(* CODESYS project State Machine.library
   Title: State Machine Twincat
   Version: 1.0.0.4
   Placeholder: State Machine Twincat
   Company: Home

Project tree, tasks and I/O mapping:
  libraries: Tc2_Standard, * (Beckhoff Automation GmbH); Tc2_System, * (Beckhoff Automation GmbH); Tc3_Module, * (Beckhoff Automation GmbH)
  DUTs/
    Actuators/
      TwoPos/
        data type E_TwoPosActuator_Fault
        data type E_TwoPosActuator_State
        data type ST_TwoPosActuator_Cfg
        data type ST_TwoPosActuator_HMI
        data type ST_TwoPosActuator_IO
        data type ST_TwoPosActuator_Sts
    Permissives/
      data type ST_PermIntlk_cfg
      data type ST_PermIntlk_HMI
      data type ST_PermIntlk_sts
    State Machine/
      data type E_SM_State
      data type SM_HMI
      data type SM_HMI_cfg
      data type SM_HMI_ocmd
      data type SM_HMI_sts
      data type ST_SM_Commands
      data type ST_SM_Conditions
      data type ST_SM_Internal
      data type ST_SM_PermissionGroups
      data type ST_SM_Permissions
      data type ST_SM_Status
      data type ST_SM_StepInfo
    Steps/
      data type ActiveStep
  GVLs/
  POUs/
    function block FB_Permissives [ST]
    function block FB_SequenceStep [ST]
    function block FB_StateMachine [ST]
    function block FB_TwoPosActuator [ST]
  VISUs/
*)

// DUTs/Actuators/TwoPos/E_TwoPosActuator_Fault
TYPE E_TwoPosActuator_Fault :
(
    None := 0,
    AdvanceTimeout := 1,
    RetractTimeout := 2,
    BothFeedbackOn := 3,
    UndefinedState := 4,
    PermissivesNotOK := 5,
    ConflictingCommands := 6,
    NoFeedback := 7
);
END_TYPE

// DUTs/Actuators/TwoPos/E_TwoPosActuator_State
TYPE E_TwoPosActuator_State :
(
    Undefined := 0,
    Retracted := 1,
    Advancing := 2,
    Advanced := 3,
    Retracting := 4,
    Fault := 5
);
END_TYPE

// DUTs/Actuators/TwoPos/ST_TwoPosActuator_Cfg
TYPE ST_TwoPosActuator_Cfg :
STRUCT
    cfgAdvTimeoutS : INT := 5;          // Advance timeout in seconds
    cfgRetTimeoutS : INT := 5;          // Retract timeout in seconds
    cfgHoldAtAdvanced : BOOL := FALSE;  // Hold valve energized when advanced
    cfgHoldAtRetracted : BOOL := FALSE; // Hold valve energized when retracted
END_STRUCT
END_TYPE

// DUTs/Actuators/TwoPos/ST_TwoPosActuator_HMI
TYPE ST_TwoPosActuator_HMI :
STRUCT
    // Status information for HMI
    sts : ST_TwoPosActuator_Sts;
    
    // Configuration from HMI
    cfg : ST_TwoPosActuator_Cfg;
    
    // Human-readable strings for HMI display
    stateString : STRING(80);      // Current state as text
    faultString : STRING(80);      // Current fault as text
    lastFaultString : STRING(80);  // Last fault as text
    
    // Operator commands from HMI
    ocmdAdvance : BOOL;         // Operator command to advance
    ocmdRetract : BOOL;         // Operator command to retract
    ocmdAllOff : BOOL;          // Operator command to turn all outputs off
    ocmdReset : BOOL;           // Operator command to reset fault
    
    // Permissive information for HMI
    advancePerms : ST_PermIntlk_HMI;  // Advance permissives
    retractPerms : ST_PermIntlk_HMI;  // Retract permissives
END_STRUCT
END_TYPE

// DUTs/Actuators/TwoPos/ST_TwoPosActuator_IO
TYPE ST_TwoPosActuator_IO :
STRUCT
    // Input feedbacks from field
    inFbkAdvanced AT %I* : BOOL;       // Advanced position feedback
    inFbkRetracted AT %I* : BOOL;      // Retracted position feedback
    
    // Output commands to field
    outValveAdvance AT %Q* : BOOL;     // Advance valve command
    outValveRetract AT %Q* : BOOL;     // Retract valve command
END_STRUCT
END_TYPE

// DUTs/Actuators/TwoPos/ST_TwoPosActuator_Sts
TYPE ST_TwoPosActuator_Sts :
STRUCT
    state : E_TwoPosActuator_State;     // Current state of actuator
    stsAdvanced : BOOL;                 // TRUE when actuator is advanced
    stsRetracted : BOOL;                // TRUE when actuator is retracted
    stsMoving : BOOL;                   // TRUE when actuator is in motion
    stsFaulted : BOOL;                  // TRUE when actuator is faulted
    faultCode : E_TwoPosActuator_Fault; // Current fault code
    lastFaultCode : E_TwoPosActuator_Fault; // Last fault code for diagnostics
    osAdvanced : BOOL;                  // One-shot when reaching advanced position
    osRetracted : BOOL;                 // One-shot when reaching retracted position
END_STRUCT
END_TYPE

// DUTs/Permissives/ST_PermIntlk_cfg
TYPE ST_PermIntlk_cfg :
STRUCT
    Name : STRING(80);                      // Name for the entire permissive set
    Desc : ARRAY [0..15] OF STRING(80);       // Descriptions for each bit
    BypassPermissives : INT;                  // Bypass bits: if a bit is 1, that permissive is bypassed
END_STRUCT
END_TYPE

// DUTs/Permissives/ST_PermIntlk_HMI
TYPE ST_PermIntlk_HMI :
STRUCT
	sts : ST_PermIntlk_sts;
	cfg : ST_PermIntlk_cfg;
END_STRUCT
END_TYPE

// DUTs/Permissives/ST_PermIntlk_sts
TYPE ST_PermIntlk_sts :
STRUCT
    PermIntlk : INT;    // Computed bitwise permissive status (each bit 1 = OK)
    OK        : BOOL;   // Overall status (TRUE if all required bits are OK)
END_STRUCT
END_TYPE

// DUTs/State Machine/E_SM_State
(* State Machine Enumeration *)
TYPE E_SM_State :
(
    STATE_IDLE := 0,
    STATE_RUNNING := 1,
    STATE_STOPPING := 2,
    STATE_HOMING := 4,
    STATE_ABORTING := 8,
    STATE_HOMED := 16,
    STATE_STOPPED := 32,
    STATE_ABORTED := 64,
    STATE_COMPLETE := 128,
    STATE_PAUSING := 256,
    STATE_PAUSED := 512,
    STATE_PROCEEDING := 1024
);
END_TYPE

// DUTs/State Machine/SM_HMI
TYPE SM_HMI :
STRUCT
  cfg : SM_HMI_cfg;
  ocmd : SM_HMI_ocmd;
  sts : SM_HMI_sts;
  NextStatePerms : ST_PermIntlk_HMI;
  ActiveStepHMI : ST_PermIntlk_HMI;
END_STRUCT
END_TYPE

// DUTs/State Machine/SM_HMI_cfg
TYPE SM_HMI_cfg :
STRUCT
  Name : STRING(40);
  HomePerm : ST_PermIntlk_HMI;
  StartPerm : ST_PermIntlk_HMI;
  ProceedPerm : ST_PermIntlk_HMI;
  AutoIntlk : ST_PermIntlk_HMI;
END_STRUCT
END_TYPE

// DUTs/State Machine/SM_HMI_ocmd
TYPE SM_HMI_ocmd :
STRUCT
  Abort : BOOL;
  Home : BOOL;
  Start : BOOL;
  Stop : BOOL;
  Pause : BOOL;
  Proceed : BOOL;
  Retry : BOOL;
  ActiveStatePermBypass : BOOL;
END_STRUCT
END_TYPE

// DUTs/State Machine/SM_HMI_sts
TYPE SM_HMI_sts :
STRUCT
  Automatic : BOOL;
  Manual : BOOL;
  StepMode : BOOL;
  Homing : BOOL;
  Homed : BOOL;
  Running : BOOL;
  Complete : BOOL;
  Stopping : BOOL;
  Stopped : BOOL;
  Aborting : BOOL;
  Aborted : BOOL;
  Pausing : BOOL;
  Paused : BOOL;
  Proceeding : BOOL;
  Faulted : BOOL;
  ChildFaulted : BOOL;
  ReadyToHome : BOOL;
  ReadyToProceed : BOOL;
  ReadyToStart : BOOL;
  AutoStartRequest : BOOL;
  AutoCycleRequest : BOOL;
  Blocked : BOOL;
  Starved : BOOL;
  Mode : DINT;
  Step : DINT;
  NextStep : DINT;
  ReturnNextStep : DINT;
END_STRUCT
END_TYPE

// DUTs/State Machine/ST_SM_Commands
(* Commands Structure - Groups all command inputs *)
TYPE ST_SM_Commands :
STRUCT
    Abort : BOOL;
    CompleteState : BOOL;
    Home : BOOL;
    Pause : BOOL;
    Proceed : BOOL;
    Retry : BOOL;
    Start : BOOL;
    Stop : BOOL;
END_STRUCT
END_TYPE

// DUTs/State Machine/ST_SM_Conditions
(* Conditions Structure - Groups process condition inputs *)
TYPE ST_SM_Conditions :
STRUCT
    Blocked : DINT;
    Starved : DINT;
END_STRUCT
END_TYPE

// DUTs/State Machine/ST_SM_Internal
(* Internal State Structure *)
TYPE ST_SM_Internal :
STRUCT
    PauseStep : ActiveStep;
    PreviousState : DINT;
    TimerReset : BOOL;
    LsOdd : DINT;
    ONS : DINT;
    StepHistoryMax : DINT;
END_STRUCT
END_TYPE

// DUTs/State Machine/ST_SM_PermissionGroups
(* Permission Group Handlers *)
TYPE ST_SM_PermissionGroups :
STRUCT
    AutoIntlk : ST_PermIntlk_HMI;
    HomePerm : ST_PermIntlk_HMI;
    ProceedPerm : ST_PermIntlk_HMI;
    StartPerm : ST_PermIntlk_HMI;
END_STRUCT
END_TYPE

// DUTs/State Machine/ST_SM_Permissions
(* Permissions Status Structure *)
TYPE ST_SM_Permissions :
STRUCT
    AutoIntlkOK : BOOL;
    HomePermOK : BOOL;
    ProceedPermOK : BOOL;
    StartPermOK : BOOL;
END_STRUCT
END_TYPE

// DUTs/State Machine/ST_SM_Status
(* Status Structure - Groups all status outputs *)
TYPE ST_SM_Status :
STRUCT
    Aborted : BOOL;
    Aborting : BOOL;
    ActiveState : BOOL;
    AutoCycleRequest : BOOL;
    Automatic : BOOL;
    AutoStartRequest : BOOL;
    Blocked : BOOL;
    Complete : BOOL;
    Faulted : BOOL;
    Homed : BOOL;
    Homing : BOOL;
    Manual : BOOL;
    Mode : DINT;
    Paused : BOOL;
    Pausing : BOOL;
    Proceeding : BOOL;
    ReadyToHome : BOOL;
    ReadyToProceed : BOOL;
    ReadyToStart : BOOL;
    Running : BOOL;
    Starved : BOOL;
    Stopped : BOOL;
    Stopping : BOOL;
    SubmoduleFaulted : BOOL;
    WaitingState : BOOL;
END_STRUCT
END_TYPE

// DUTs/State Machine/ST_SM_StepInfo
(* Step Information Structure *)
TYPE ST_SM_StepInfo :
STRUCT
    CurrentStep : DINT;
    NextStep : DINT;
    ReturnNextStep : DINT;
    ReturnState : DINT;  // Changed from enum to DINT for compatibility
    LastState : DINT;    // Changed from enum to DINT for compatibility
    CurrentState : DINT; // Changed from enum to DINT for compatibility
    StateString : STRING(40);
    StepTimerSeconds : REAL;
END_STRUCT
END_TYPE

// DUTs/Steps/ActiveStep
TYPE ActiveStep  :
STRUCT
  Step : DINT;
  StatusStepFaulted : BOOL;
  PermsHMI : ST_PermIntlk_cfg;
END_STRUCT
END_TYPE

// POUs/FB_Permissives
{attribute 'hide_all_locals'}
FUNCTION_BLOCK FB_Permissives
VAR_INPUT
    inPermissives : INT;           // Real-world permissive bits from hardware/sensors
    cfg           : ST_PermIntlk_cfg; // Configuration: name, bit descriptions, and bypass settings
END_VAR
VAR_OUTPUT PERSISTENT
    stsOK       : BOOL;            // Overall computed status (TRUE if all required permissives are OK)
    PermStatus  : INT;             // Bitwise computed permissive status (each bit set to 1 means that bit is OK)
END_VAR
VAR
    i         : INT;
    localStatus : INT;             // Local working variable for status
END_VAR

// Clear local status at start of each cycle
localStatus := 0;

// Loop over bits 0 to 15
FOR i := 0 TO 15 DO
    // Check if bypass is active for this bit (bypass bits are in cfg)
    IF (cfg.BypassPermissives AND SHL(1, i)) <> 0 THEN
        // Bypassed: treat this bit as OK
        localStatus := localStatus OR SHL(1, i);
    ELSE
        // Otherwise, if the real permissive bit is set, mark it as OK
        IF (inPermissives AND SHL(1, i)) <> 0 THEN
            localStatus := localStatus OR SHL(1, i);
        END_IF;
    END_IF;
END_FOR

// Save computed status to output variable
PermStatus := localStatus;

// Overall status: if all 16 bits are OK then stsOK is TRUE.
stsOK := (localStatus = -1);

END_FUNCTION_BLOCK

// POUs/FB_SequenceStep
{attribute 'hide_all_locals'}
FUNCTION_BLOCK FB_SequenceStep
VAR_INPUT
    inpStep              : DINT;  // Current step number (from sequence controller)
    cfgStep              : DINT;  // This FB's step number (step ID)
    cfgNextStep          : DINT;  // Next step if permissives are OK
    inpStepTimerSeconds  : DINT;  // Step timer value (managed externally)
    inpRetry             : BOOL;  // External retry command (to reset fault)
    inpStepPermissives   : INT;   // Actual permissive bits (from sensors, PLC, etc.)
    cfgStepTimeout       : INT;   // Timeout configuration (in seconds)
	inpFaultStep         : BOOL;  // Fault conditions outside of timeout 
END_VAR

VAR_IN_OUT
    ActiveStep           : ActiveStep; 
    // ActiveStep holds:
    //   Step              : DINT;  (current step number)
    //   StatusStepFaulted : BOOL;  (fault flag)
    //   PermsHMI          : ST_PermIntlk_cfg; (permissive configuration: Name, Desc, BypassPermissives)
END_VAR

VAR_OUTPUT
    outStepActive         : BOOL;  // TRUE when this step is active
    outStepActiveOS       : BOOL;  // One-shot rising pulse when step becomes active
    outFaultedStepActive  : BOOL;  // TRUE when this step is faulted
    outFaultedStepActiveOS: BOOL;  // One-shot rising pulse when a fault occurs
    outActiveStepTimedOut : BOOL;  // TRUE when the step times out
    outNextStep           : DINT;  // The next step number in sequence
END_VAR

VAR
    Step_P_Perm    : FB_Permissives; // Instance for permissives check
    rTrig_Activate : R_TRIG;         // Rising edge detector for step activation
    rTrig_Fault    : R_TRIG;         // Rising edge detector for fault detection
    rTrig_Retry    : R_TRIG;         // Rising edge detector for retry detection
END_VAR

// 1. Evaluate Permissives using FB_Permissives
Step_P_Perm.inPermissives := inpStepPermissives;
Step_P_Perm.cfg           := ActiveStep.PermsHMI;
Step_P_Perm();  // Execute permissives check

// 2. Update the ActiveStep with the current step
ActiveStep.Step := inpStep;

// 3. Determine if this step is active (active when inpStep equals cfgStep)
outStepActive := (inpStep = cfgStep);

// 4. Generate a one-shot pulse for step activation (rising edge)
rTrig_Activate.CLK := outStepActive;
rTrig_Activate();
outStepActiveOS := rTrig_Activate.Q;


// 5. Timeout Handling: If the externally managed timer exceeds the configured timeout, flag as timed out
IF 
(cfgStepTimeout <> 0 ) AND // cfgStepTimeout = 0 for no timeout fault
(inpStepTimerSeconds > cfgStepTimeout) 
THEN
    outActiveStepTimedOut := TRUE;
ELSE
    outActiveStepTimedOut := FALSE;
END_IF;

// 6. Fault Condition:
// A fault occurs if the step is active, the step has timed out, and the permissives are NOT OK.
IF outStepActive AND outActiveStepTimedOut AND (NOT Step_P_Perm.stsOK) 
OR inpFaultStep
THEN
    ActiveStep.StatusStepFaulted := TRUE;
END_IF;

// 7. Set the fault output based on the ActiveStep fault status
outFaultedStepActive := ActiveStep.StatusStepFaulted;

// 8. Generate a one-shot pulse for fault detection (rising edge)
rTrig_Fault.CLK := outFaultedStepActive;
rTrig_Fault();
outFaultedStepActiveOS := rTrig_Fault.Q;

// 9. Retry Logic: if a retry command is detected (rising edge on inpRetry) while faulted, clear the fault flag
rTrig_Retry.CLK := inpRetry;
rTrig_Retry();
IF rTrig_Retry.Q AND outFaultedStepActive THEN
    ActiveStep.StatusStepFaulted := FALSE;
END_IF;

// 10. Determine the next step:
// - If the step is faulted, set outNextStep to cfgStep + 1 (fault-handling step).
// - Else if the permissives are OK and the step is active, set outNextStep to cfgNextStep.
// - Otherwise, remain on the current step.
IF outFaultedStepActive THEN
    outNextStep := cfgStep + 1;
ELSIF Step_P_Perm.stsOK AND outStepActive THEN
    outNextStep := cfgNextStep;
ELSE
    outNextStep := inpStep;
END_IF;

END_FUNCTION_BLOCK

// POUs/FB_StateMachine
{attribute 'hide_all_locals'} // Hides all local variables
FUNCTION_BLOCK FB_StateMachine
VAR_INPUT
    EnableIn : BOOL;                     // Enable input for the function block
    cfgAutoRun : BOOL;                   // Configuration for auto-run capability
    inpAutoIntlk : INT := -1;            // Auto interlock input bits
    inpBlockedCondition : DINT;          // Blocked condition input
    inpHomePerm : INT := -1;             // Home permission input bits
    inpProceedPerm : INT := -1;          // Proceed permission input bits
    inpStartPerm : INT := -1;            // Start permission input bits
    inpStarvedCondition : DINT;          // Starved condition input
    inpSubmoduleFaulted : BOOL;          // Submodule fault indicator
END_VAR

VAR_OUTPUT
    EnableOut : BOOL;                    // Enable output for the function block
    outRetry : BOOL;                     // Retry output signal
    Status : ST_SM_Status;               // Status outputs (grouped)
    Permissions : ST_SM_Permissions;     // Permission status outputs (grouped)
    StepInfo : ST_SM_StepInfo;           // Step information (grouped)
    ConditionStatus : ST_SM_Conditions;  // Condition status (grouped)
END_VAR

VAR CONSTANT
    internalClearStep : ActiveStep;      // Constant for clearing a step
    EmptyHMIPerm : ST_PermIntlk_HMI;     // Empty HMI permissions structure
    
    // State constants
    STATE_IDLE : INT := 0;
    STATE_RUNNING : INT := 1;
    STATE_STOPPING : INT := 2;
    STATE_HOMING : INT := 4;
    STATE_ABORTING : INT := 8;
    STATE_HOMED : INT := 16;
    STATE_STOPPED : INT := 32;
    STATE_ABORTED : INT := 64;
    STATE_COMPLETE : INT := 128;
    STATE_PAUSING : INT := 256;
    STATE_PAUSED : INT := 512;
    STATE_PROCEEDING : INT := 1024;

    // Step range constants for sequence inference
    HOMING_MIN   : DINT := 1000; HOMING_MAX   : DINT := 1999;
    RUNNING_MIN  : DINT := 3000; RUNNING_MAX  : DINT := 3999;
    STOPPING_MIN : DINT := 2000; STOPPING_MAX : DINT := 2999;
    ABORTING_MIN : DINT := 5000; ABORTING_MAX : DINT := 5999;
    PAUSING_MIN  : DINT := 4000; PAUSING_MAX  : DINT := 4999;
    PROCEEDING_MIN : DINT := 6000; PROCEEDING_MAX : DINT := 6999;
END_VAR

VAR
    // Command request tracking
    CommandsRequested : ST_SM_Commands;  // Track command requests
    RetryComplete : BOOL;                // Flag for retry completion
    
    // Timer
    StepTimer : TON;                     // Step timer
    
    // Edge detection for commands
    R_TRIG_1 : R_TRIG;                  // For step transition
    R_TRIG_2 : R_TRIG;                  // For command retry
    R_TRIG_3 : R_TRIG;                  // For HMI retry
    R_TRIG_4 : R_TRIG;                  // For state transitions
    R_TRIG_5 : R_TRIG;                  // For sequence complete inference
    
    // Internal state tracking
    PauseStep : ActiveStep;              // Store step during pause
    PreviousState : DINT;                // Previous state
    PreviousStep : DINT;                 // Previous step for reference
    TimerReset : BOOL;                   // Flag to reset timer
    LsOdd : DINT;                        // Odd step check for fault detection
    ONS : DINT;                          // General one-shot
    StepHistoryMax : DINT;               // Step history maximum
    ReturnState : DINT;                  // Return state after pause
    ReturnNextStep : DINT;               // Return next step after pause
    
    // Permission handlers
    internalAutoIntlk : FB_Permissives;       // Auto interlock handler
    internalHomePerm : FB_Permissives;        // Home permission handler
    internalProceedPerm : FB_Permissives;     // Proceed permission handler
    internalStartPerm : FB_Permissives;       // Start permission handler
    
    // Configuration for permission handlers
    homePermCfg : ST_PermIntlk_cfg;      // Configuration for home permission handler
    startPermCfg : ST_PermIntlk_cfg;     // Configuration for start permission handler
    proceedPermCfg : ST_PermIntlk_cfg;   // Configuration for proceed permission handler
    autoIntlkCfg : ST_PermIntlk_cfg;     // Configuration for auto interlock handler
    
    // HMI data structures for permissions
    internalAutoIntlk_HMI : ST_PermIntlk_HMI;  // Auto interlock HMI structure
    internalHomePerm_HMI : ST_PermIntlk_HMI;   // Home permission HMI structure
    internalProceedPerm_HMI : ST_PermIntlk_HMI; // Proceed permission HMI structure
    internalStartPerm_HMI : ST_PermIntlk_HMI;  // Start permission HMI structure
    
    // Temp variables for step detection
    stepIsZero : BOOL;                   // Flag for zero step
    retryCmdActive : BOOL;               // Flag for retry command
    retryHmiActive : BOOL;               // Flag for HMI retry
    transitionActive : BOOL;             // Flag for state transition
    seqDone : BOOL;                      // Inferred sequence completion
END_VAR

VAR_IN_OUT 
    HMI : SM_HMI;                        // HMI interface
    CurrentStep : ActiveStep;            // Current active step
	NextStep : DINT;                     // Next step to transition to
	Commands : ST_SM_Commands;           // Command inputs (grouped)
END_VAR


//-----------------------------------------------------------------------------
// Main Implementation
//-----------------------------------------------------------------------------
EnableOut := EnableIn;

// Only execute if enabled
IF EnableIn THEN
    //-------------------------------------------------------------------------
    // Process permissions for different states
    //-------------------------------------------------------------------------
    
    // Update configuration from HMI
    homePermCfg := internalHomePerm_HMI.cfg;
    startPermCfg := internalStartPerm_HMI.cfg;
    proceedPermCfg := internalProceedPerm_HMI.cfg;
    autoIntlkCfg := internalAutoIntlk_HMI.cfg;
    
    // Home permission evaluation
    internalHomePerm(
        inPermissives := inpHomePerm,
        cfg := homePermCfg
    );
    Permissions.HomePermOK := internalHomePerm.stsOK;
    internalHomePerm_HMI.sts.OK := internalHomePerm.stsOK;
    internalHomePerm_HMI.sts.PermIntlk := internalHomePerm.PermStatus;
    
    // Start permission evaluation
    internalStartPerm(
        inPermissives := inpStartPerm,
        cfg := startPermCfg
    );
    Permissions.StartPermOK := internalStartPerm.stsOK;
    internalStartPerm_HMI.sts.OK := internalStartPerm.stsOK;
    internalStartPerm_HMI.sts.PermIntlk := internalStartPerm.PermStatus;
    
    // Proceed permission evaluation
    internalProceedPerm(
        inPermissives := inpProceedPerm,
        cfg := proceedPermCfg
    );
    Permissions.ProceedPermOK := internalProceedPerm.stsOK;
    internalProceedPerm_HMI.sts.OK := internalProceedPerm.stsOK;
    internalProceedPerm_HMI.sts.PermIntlk := internalProceedPerm.PermStatus;
    
    // Auto interlock evaluation
    internalAutoIntlk(
        inPermissives := inpAutoIntlk,
        cfg := autoIntlkCfg
    );
    Permissions.AutoIntlkOK := internalAutoIntlk.stsOK;
    internalAutoIntlk_HMI.sts.OK := internalAutoIntlk.stsOK;
    internalAutoIntlk_HMI.sts.PermIntlk := internalAutoIntlk.PermStatus;
    
    //-------------------------------------------------------------------------
    // Ready state calculations
    //-------------------------------------------------------------------------
    
    // Ready to Home: Stopped or Aborted + Home permissions OK + Auto interlock OK
    Status.ReadyToHome := (Status.Stopped OR Status.Aborted) AND 
                          Permissions.HomePermOK AND 
                          Permissions.AutoIntlkOK;
    
    // Ready to Start: (Homed or Complete) + Start permissions OK + Auto interlock OK + Not auto-start requested
    Status.ReadyToStart := (Status.Homed OR Status.Complete) AND 
                          Permissions.StartPermOK AND 
                          Permissions.AutoIntlkOK AND 
                          NOT Status.AutoStartRequest;
    
    // Ready to Proceed: Paused + Proceed permissions OK + Auto interlock OK
    Status.ReadyToProceed := Status.Paused AND 
                            Permissions.ProceedPermOK AND 
                            Permissions.AutoIntlkOK;

    //-------------------------------------------------------------------------
    // Clear Active Step if in waiting state
    //-------------------------------------------------------------------------
    IF Status.Homed OR Status.Complete OR Status.Stopped OR Status.Aborted THEN
        CurrentStep := internalClearStep;
    END_IF;
    
    // Clear pause step on proceeding or aborting
    transitionActive := Status.Proceeding OR Status.Aborting;
    R_TRIG_4(CLK := transitionActive);
    IF R_TRIG_4.Q THEN
        PauseStep := internalClearStep;
    END_IF;
    
    //-------------------------------------------------------------------------
    // Auto-start request logic
    //-------------------------------------------------------------------------
    
    // Auto start request handling
    Status.AutoStartRequest := CommandsRequested.Start AND NOT Permissions.StartPermOK;
    
    // Auto cycle request for auto-run when complete
    Status.AutoCycleRequest := cfgAutoRun AND Status.Complete AND NOT Permissions.StartPermOK;
    
    //-------------------------------------------------------------------------
    // Remember last state before change
    //-------------------------------------------------------------------------
    PreviousState := StepInfo.CurrentState;
    
    //-------------------------------------------------------------------------
    // Process command requests
    //-------------------------------------------------------------------------
    
    // Complete State Request
    IF Commands.CompleteState THEN
        CommandsRequested.CompleteState := TRUE;
        Commands.CompleteState := FALSE;  // Reset command
        // Clear other requests
        CommandsRequested.Start := FALSE;
        CommandsRequested.Abort := FALSE;
        CommandsRequested.Pause := FALSE;
        CommandsRequested.Home := FALSE;
        CommandsRequested.Proceed := FALSE;
        CommandsRequested.Stop := FALSE;
    END_IF;
    
    // Start Request
    IF Commands.Start OR HMI.ocmd.Start THEN
        IF Permissions.AutoIntlkOK AND Permissions.StartPermOK AND (Status.Homed OR Status.Complete) THEN
            CommandsRequested.Start := TRUE;
        END_IF;
        
        IF CommandsRequested.Start AND (Status.Homed OR Status.Complete OR Status.Stopped) OR Status.AutoStartRequest THEN
            CommandsRequested.Start := TRUE;
        END_IF;
        
        // Clear command signals
        IF Commands.Start THEN
            Commands.Start := FALSE;
        END_IF;
        
        IF HMI.ocmd.Start THEN
            HMI.ocmd.Start := FALSE;
        END_IF;
    END_IF;
    
    // Clear other requests if Start is requested
    IF CommandsRequested.Start THEN
        CommandsRequested.Abort := FALSE;
        CommandsRequested.Pause := FALSE;
        CommandsRequested.Home := FALSE;
        CommandsRequested.Proceed := FALSE;
        CommandsRequested.Stop := FALSE;
        CommandsRequested.CompleteState := FALSE;
    END_IF;
    
    // Auto-run handling
    IF cfgAutoRun AND Permissions.AutoIntlkOK AND Permissions.StartPermOK AND Status.Complete THEN
        CommandsRequested.Start := TRUE;
    END_IF;
    
    // Home Request
    IF Commands.Home OR HMI.ocmd.Home THEN
        IF (Status.Stopped OR Status.Aborted) AND Permissions.HomePermOK AND Permissions.AutoIntlkOK THEN
            CommandsRequested.Home := TRUE;
        END_IF;
        
        // Clear other requests
        CommandsRequested.Abort := FALSE;
        CommandsRequested.Pause := FALSE;
        CommandsRequested.Proceed := FALSE;
        CommandsRequested.Start := FALSE;
        CommandsRequested.Stop := FALSE;
        CommandsRequested.CompleteState := FALSE;
        
        // Clear command signals
        IF Commands.Home THEN
            Commands.Home := FALSE;
        END_IF;
        
        IF HMI.ocmd.Home THEN
            HMI.ocmd.Home := FALSE;
        END_IF;
    END_IF;
    
    // Pause Request
    IF Commands.Pause OR HMI.ocmd.Pause THEN
        CommandsRequested.Pause := TRUE;
        
        // Clear other requests
        CommandsRequested.Abort := FALSE;
        CommandsRequested.Home := FALSE;
        CommandsRequested.Proceed := FALSE;
        CommandsRequested.Start := FALSE;
        CommandsRequested.Stop := FALSE;
        CommandsRequested.CompleteState := FALSE;
        
        // Clear command signals
        IF Commands.Pause THEN
            Commands.Pause := FALSE;
        END_IF;
        
        IF HMI.ocmd.Pause THEN
            HMI.ocmd.Pause := FALSE;
        END_IF;
    END_IF;
    
    // Proceed Request
    IF Commands.Proceed OR HMI.ocmd.Proceed THEN
        IF Permissions.ProceedPermOK AND Permissions.AutoIntlkOK THEN
            CommandsRequested.Proceed := TRUE;
        END_IF;
        
        // Clear other requests
        CommandsRequested.Abort := FALSE;
        CommandsRequested.Home := FALSE;
        CommandsRequested.Pause := FALSE;
        CommandsRequested.Start := FALSE;
        CommandsRequested.Stop := FALSE;
        CommandsRequested.CompleteState := FALSE;
        
        // Clear command signals
        IF Commands.Proceed THEN
            Commands.Proceed := FALSE;
        END_IF;
        
        IF HMI.ocmd.Proceed THEN
            HMI.ocmd.Proceed := FALSE;
        END_IF;
    END_IF;
    
    // Stop Request
    IF Commands.Stop OR HMI.ocmd.Stop THEN
        CommandsRequested.Stop := TRUE;
        
        // Clear other requests
        CommandsRequested.Abort := FALSE;
        CommandsRequested.Home := FALSE;
        CommandsRequested.Proceed := FALSE;
        CommandsRequested.Start := FALSE;
        CommandsRequested.Pause := FALSE;
        CommandsRequested.CompleteState := FALSE;
        
        // Clear command signals
        IF Commands.Stop THEN
            Commands.Stop := FALSE;
        END_IF;
        
        IF HMI.ocmd.Stop THEN
            HMI.ocmd.Stop := FALSE;
        END_IF;
    END_IF;
    
    // Abort Request
    IF Commands.Abort OR HMI.ocmd.Abort THEN
        CommandsRequested.Abort := TRUE;
        
        // Clear other requests
        CommandsRequested.Stop := FALSE;
        CommandsRequested.Home := FALSE;
        CommandsRequested.Proceed := FALSE;
        CommandsRequested.Start := FALSE;
        CommandsRequested.Pause := FALSE;
        CommandsRequested.CompleteState := FALSE;
        
        // Clear command signals
        IF Commands.Abort THEN
            Commands.Abort := FALSE;
        END_IF;
        
        IF HMI.ocmd.Abort THEN
            HMI.ocmd.Abort := FALSE;
        END_IF;
    END_IF;
    
    //-------------------------------------------------------------------------
    // Sequence completion inference
    //-------------------------------------------------------------------------
    // If in an active state with a defined sequence range and the sequence
    // drives NextStep to 0 while the current step is within that state's
    // range, infer completion and trigger CompleteState internally.
    seqDone := FALSE;
    IF Status.Homing THEN
        seqDone := (StepInfo.CurrentStep >= HOMING_MIN) AND (StepInfo.CurrentStep <= HOMING_MAX) AND (NextStep = 0);
    ELSIF Status.Running THEN
        seqDone := (StepInfo.CurrentStep >= RUNNING_MIN) AND (StepInfo.CurrentStep <= RUNNING_MAX) AND (NextStep = 0);
    ELSIF Status.Stopping THEN
        seqDone := (StepInfo.CurrentStep >= STOPPING_MIN) AND (StepInfo.CurrentStep <= STOPPING_MAX) AND (NextStep = 0);
    ELSIF Status.Aborting THEN
        seqDone := (StepInfo.CurrentStep >= ABORTING_MIN) AND (StepInfo.CurrentStep <= ABORTING_MAX) AND (NextStep = 0);
    ELSIF Status.Pausing THEN
        seqDone := (StepInfo.CurrentStep >= PAUSING_MIN) AND (StepInfo.CurrentStep <= PAUSING_MAX) AND (NextStep = 0);
    ELSIF Status.Proceeding THEN
        seqDone := (StepInfo.CurrentStep >= PROCEEDING_MIN) AND (StepInfo.CurrentStep <= PROCEEDING_MAX) AND (NextStep = 0);
    END_IF;

    R_TRIG_5(CLK := seqDone);
    IF R_TRIG_5.Q THEN
        CommandsRequested.CompleteState := TRUE;
    END_IF;

    //-------------------------------------------------------------------------
    // State Transitions
    //-------------------------------------------------------------------------

    // Complete to Homed
    IF CommandsRequested.CompleteState AND Status.Homing THEN
        NextStep := 0;
        StepInfo.CurrentState := STATE_HOMED;
        CommandsRequested.CompleteState := FALSE;  // Clear after transition
    END_IF;
    
    // Running to Complete
    IF CommandsRequested.CompleteState AND Status.Running THEN
        NextStep := 0;
        StepInfo.CurrentState := STATE_COMPLETE;
        CommandsRequested.CompleteState := FALSE;  // Clear after transition
    END_IF;
    
    // Running to Stopping
    IF CommandsRequested.Stop AND Status.Running THEN
        StepInfo.CurrentState := STATE_STOPPING;
    END_IF;
    
    // Stopping to Stopped
    IF CommandsRequested.CompleteState AND Status.Stopping THEN
        NextStep := 0;
        StepInfo.CurrentState := STATE_STOPPED;
        CommandsRequested.CompleteState := FALSE;  // Clear after transition
    END_IF;
    
    // Aborting to Aborted
    IF CommandsRequested.CompleteState AND Status.Aborting THEN
        NextStep := 0;
        StepInfo.CurrentState := STATE_ABORTED;
        CommandsRequested.CompleteState := FALSE;  // Clear after transition
    END_IF;
    
    // Active State to Pausing
    // Handle state transitions to Pausing and remember the state to return to
    IF CommandsRequested.Pause AND (
        Status.Homing OR Status.Stopping OR Status.Aborting OR 
        Status.Homed OR Status.Complete OR Status.Proceeding OR Status.Running) THEN
        
        // Remember the current state and next step for later return
        IF NOT (Status.Homed OR Status.Complete OR Status.Proceeding) THEN
            ReturnState := StepInfo.CurrentState;
            ReturnNextStep := NextStep;
        END_IF;
        
        // Save the current step for paused state
        IF NOT (Status.Homed OR Status.Complete OR Status.Proceeding) THEN
            PauseStep := CurrentStep;
        ELSE
            PauseStep := internalClearStep;
        END_IF;
        
        // Transition to pausing state
        StepInfo.CurrentState := STATE_PAUSING;
        NextStep := 0;
    END_IF;
    
    // Pausing to Paused
    IF CommandsRequested.CompleteState AND Status.Pausing THEN
        NextStep := 0;
        StepInfo.CurrentState := STATE_PAUSED;
        CommandsRequested.CompleteState := FALSE;  // Clear after transition
    END_IF;
    
    // Proceeding to Step before Pausing
    IF CommandsRequested.CompleteState AND Status.Proceeding THEN
        CurrentStep := PauseStep;
        NextStep := ReturnNextStep;
        StepInfo.CurrentState := ReturnState;
        CommandsRequested.CompleteState := FALSE;  // Clear after transition
    END_IF;
    
    // Homed to Running
    IF (CommandsRequested.Start OR 
        (Status.AutoStartRequest AND Permissions.StartPermOK AND Permissions.AutoIntlkOK)) AND 
        (Status.Homed OR Status.Complete) THEN
        
        NextStep := 0;
        StepInfo.CurrentState := STATE_RUNNING;
        CommandsRequested.Start := FALSE;
    END_IF;
    
    // Homed to Stopped
    IF CommandsRequested.Stop AND Status.Homed THEN
        NextStep := 0;
        StepInfo.CurrentState := STATE_STOPPED;
    END_IF;
    
    // Complete to Stopped
    IF CommandsRequested.Stop AND Status.Complete THEN
        NextStep := 0;
        StepInfo.CurrentState := STATE_STOPPED;
    END_IF;
    
    // Stopped or Aborted to Homing
    IF CommandsRequested.Home AND (Status.Stopped OR Status.Aborted) THEN
        NextStep := 0;
        StepInfo.CurrentState := STATE_HOMING;
    END_IF;
    
    // Paused to Proceeding
    IF CommandsRequested.Proceed AND Status.Paused THEN
        NextStep := 0;
        StepInfo.CurrentState := STATE_PROCEEDING;
    END_IF;
    
    // Abort (from any state except Stopped/Aborted/Aborting)
    IF CommandsRequested.Abort AND NOT (Status.Stopped OR Status.Aborted OR Status.Aborting) THEN
        NextStep := 0;
        StepInfo.CurrentState := STATE_ABORTING;
    END_IF;
    
    //-------------------------------------------------------------------------
    // Save last state when changing
    //-------------------------------------------------------------------------
    IF StepInfo.CurrentState <> PreviousState THEN
        StepInfo.LastState := PreviousState;
    END_IF;
    
    //-------------------------------------------------------------------------
    // Update status flags based on current state
    //-------------------------------------------------------------------------
    // Reset all status flags first
    Status.Running := FALSE;
    Status.Stopping := FALSE;
    Status.Homing := FALSE;
    Status.Aborting := FALSE;
    Status.Homed := FALSE;
    Status.Stopped := FALSE;
    Status.Aborted := FALSE;
    Status.Complete := FALSE;
    Status.Pausing := FALSE;
    Status.Paused := FALSE;
    Status.Proceeding := FALSE;
    
    // Set corresponding status flag based on current state
    CASE StepInfo.CurrentState OF
        STATE_RUNNING:
            Status.Running := TRUE;
            StepInfo.StateString := 'Running';
        
        STATE_STOPPING:
            Status.Stopping := TRUE;
            StepInfo.StateString := 'Stopping';
        
        STATE_HOMING:
            Status.Homing := TRUE;
            StepInfo.StateString := 'Homing';
        
        STATE_ABORTING:
            Status.Aborting := TRUE;
            StepInfo.StateString := 'Aborting';
        
        STATE_HOMED:
            Status.Homed := TRUE;
            StepInfo.StateString := 'Homed';
        
        STATE_STOPPED:
            Status.Stopped := TRUE;
            StepInfo.StateString := 'Stopped';
        
        STATE_ABORTED:
            Status.Aborted := TRUE;
            StepInfo.StateString := 'Aborted';
        
        STATE_COMPLETE:
            Status.Complete := TRUE;
            StepInfo.StateString := 'Complete';
        
        STATE_PAUSING:
            Status.Pausing := TRUE;
            StepInfo.StateString := 'Pausing';
        
        STATE_PAUSED:
            Status.Paused := TRUE;
            StepInfo.StateString := 'Paused';
        
        STATE_PROCEEDING:
            Status.Proceeding := TRUE;
            StepInfo.StateString := 'Proceeding';
    END_CASE;
    
    // Set the active/waiting state flags
    Status.WaitingState := Status.Homed OR Status.Complete OR Status.Stopped OR Status.Paused OR Status.Aborted;
    Status.ActiveState := Status.Homing OR Status.Running OR Status.Stopping OR Status.Pausing OR Status.Proceeding OR Status.Aborting;
    
    // Set mode (0 = Manual, 1 = Automatic)
    IF Status.Stopped OR Status.Aborted OR Status.Paused THEN
        Status.Mode := 0;
        Status.Manual := TRUE;
        Status.Automatic := FALSE;
    ELSE
        Status.Mode := 1;
        Status.Manual := FALSE;
        Status.Automatic := TRUE;
    END_IF;

    //-------------------------------------------------------------------------
    // Step and timer management
    //-------------------------------------------------------------------------
    
    // Clear ActiveStep when transitioning to step 0 (when step becomes zero)
    stepIsZero := (StepInfo.CurrentStep = 0);
    R_TRIG_1(CLK := stepIsZero);
    IF R_TRIG_1.Q THEN
        CurrentStep := internalClearStep;
        // Also reset timer when entering step 0 (state transitions)
        TimerReset := TRUE;
        StepTimer(IN := FALSE, PT := T#99H);
        StepInfo.StepTimerSeconds := 0.0;  // Immediately clear the timer output
    END_IF;
    
    // Detect step change and update step - AFTER clearing logic
    IF StepInfo.CurrentStep <> NextStep THEN
        // Store previous step for reference
        PreviousStep := StepInfo.CurrentStep;
        StepInfo.CurrentStep := NextStep;
        TimerReset := TRUE;
        // Immediately reset timer when step changes
        StepTimer(IN := FALSE, PT := T#99H);
        StepInfo.StepTimerSeconds := 0.0;  // Immediately clear the timer output
    END_IF;
    
    // Synchronize shared CurrentStep.Step with internal step tracking - AFTER all step updates
    IF CurrentStep.Step <> StepInfo.CurrentStep THEN
        CurrentStep.Step := StepInfo.CurrentStep;
    END_IF;
    
    // Step timer logic
    IF NOT Status.Paused OR (Status.Paused AND CommandsRequested.CompleteState) THEN
        IF TimerReset THEN
            // Keep timer reset for one scan, then clear flag
            StepTimer(IN := FALSE, PT := T#99H);
            StepInfo.StepTimerSeconds := 0.0;  // Ensure timer value is zero during reset
            TimerReset := FALSE;
        ELSE
            // Normal timer operation
            StepTimer(IN := TRUE, PT := T#99H);
            // Convert timer value to seconds only when not resetting
            StepInfo.StepTimerSeconds := UDINT_TO_REAL(TIME_TO_UDINT(StepTimer.ET)) / 1000.0;
        END_IF;
    ELSE
        StepTimer(IN := FALSE, PT := T#99H);
        // Don't update StepTimerSeconds when paused unless transitioning
    END_IF;
    
    //-------------------------------------------------------------------------
    // Fault detection
    //-------------------------------------------------------------------------
    
    // Check if step is odd (indicates fault)
    LsOdd := StepInfo.CurrentStep MOD 2;
    Status.Faulted := LsOdd <> 0;
    
    // Submodule fault handling
    Status.SubmoduleFaulted := inpSubmoduleFaulted;
    
    //-------------------------------------------------------------------------
    // Retry logic
    //-------------------------------------------------------------------------
    
    // Retry command from command input
    retryCmdActive := Commands.Retry;
    R_TRIG_2(CLK := retryCmdActive);
    IF R_TRIG_2.Q THEN
        outRetry := TRUE;
        Commands.Retry := FALSE;
    END_IF;
    
    // Retry command from HMI
    retryHmiActive := HMI.ocmd.Retry;
    R_TRIG_3(CLK := retryHmiActive);
    IF R_TRIG_3.Q THEN
        outRetry := TRUE;
        HMI.ocmd.Retry := FALSE;
    END_IF;
    
    // Ensure retry signal stays on for at least one scan
    IF RetryComplete THEN
        outRetry := FALSE;
        RetryComplete := FALSE;
    END_IF;
    
    IF outRetry THEN
        RetryComplete := TRUE;
    END_IF;
    
    //-------------------------------------------------------------------------
    // Blocked and Starved condition handling for OEE
    //-------------------------------------------------------------------------
    
    // Reset blocked condition if not present
    IF inpBlockedCondition = 0 THEN
        ConditionStatus.Blocked := 0;
    END_IF;
    
    // Check for blocked condition in appropriate states
    IF inpBlockedCondition <> 0 AND 
       (Status.Running OR Status.Stopping OR Status.Complete OR 
        (Status.Homed AND Status.AutoStartRequest)) THEN
        
        ConditionStatus.Blocked := inpBlockedCondition;
        Status.Blocked := TRUE;
        inpBlockedCondition := 0;
    END_IF;
    
    // Reset starved condition if not present
    IF inpStarvedCondition = 0 THEN
        ConditionStatus.Starved := 0;
    END_IF;
    
    // Check for starved condition in appropriate states
    IF inpStarvedCondition <> 0 AND 
       (Status.Running OR Status.Stopping OR Status.Complete OR 
        (Status.Homed AND Status.AutoStartRequest)) THEN
        
        ConditionStatus.Starved := inpStarvedCondition;
        Status.Starved := TRUE;
        inpStarvedCondition := 0;
    END_IF;
    
    //-------------------------------------------------------------------------
    // Update HMI data
    //-------------------------------------------------------------------------
    
    // Update HMI status information
    HMI.sts.Automatic := Status.Automatic;
    HMI.sts.Manual := Status.Manual;
    HMI.sts.Homing := Status.Homing;
    HMI.sts.Homed := Status.Homed;
    HMI.sts.Running := Status.Running;
    HMI.sts.Complete := Status.Complete;
    HMI.sts.Stopping := Status.Stopping;
    HMI.sts.Stopped := Status.Stopped;
    HMI.sts.Aborting := Status.Aborting;
    HMI.sts.Aborted := Status.Aborted;
    HMI.sts.Pausing := Status.Pausing;
    HMI.sts.Paused := Status.Paused;
    HMI.sts.Proceeding := Status.Proceeding;
    HMI.sts.Faulted := Status.Faulted;
    HMI.sts.ChildFaulted := Status.SubmoduleFaulted;
    HMI.sts.ReadyToHome := Status.ReadyToHome;
    HMI.sts.ReadyToProceed := Status.ReadyToProceed;
    HMI.sts.ReadyToStart := Status.ReadyToStart;
    HMI.sts.AutoStartRequest := Status.AutoStartRequest;
    HMI.sts.AutoCycleRequest := Status.AutoCycleRequest;
    HMI.sts.Blocked := Status.Blocked;
    HMI.sts.Starved := Status.Starved;
    
    // Update permission states in HMI
    IF Status.Stopped OR Status.Aborted THEN
        HMI.NextStatePerms := internalHomePerm_HMI;
    END_IF;
    
    IF Status.Homed OR Status.Complete THEN
        HMI.NextStatePerms := internalStartPerm_HMI;
    END_IF;
    
    IF Status.Paused THEN
        HMI.NextStatePerms := internalProceedPerm_HMI;
    END_IF;
    
    // Update active step information
    IF Status.ActiveState THEN
        // Create a HMI structure with the current step's permission config
        internalHomePerm_HMI.cfg := CurrentStep.PermsHMI;
        HMI.ActiveStepHMI := internalHomePerm_HMI;
    ELSE
        HMI.ActiveStepHMI := HMI.NextStatePerms;
    END_IF;
    
ELSE
    // Reset command requests when disabled
    CommandsRequested.Start := FALSE;
    CommandsRequested.Stop := FALSE;
    CommandsRequested.Home := FALSE;
    CommandsRequested.Abort := FALSE;
    CommandsRequested.Pause := FALSE;
    CommandsRequested.Proceed := FALSE;
    CommandsRequested.CompleteState := FALSE;
END_IF;

END_FUNCTION_BLOCK

// POUs/FB_TwoPosActuator
{attribute 'hide_all_locals'} // Hides all local variables
FUNCTION_BLOCK FB_TwoPosActuator
VAR_INPUT
    EnableIn : BOOL := TRUE;            // Enable input for the function block
    inWorkingMode : BOOL := TRUE;       // Working mode: TRUE=Auto, FALSE=Manual
    
    // Program commands (automatic mode only)
    pcmdAdvance : BOOL;                 // Program command to advance
    pcmdRetract : BOOL;                 // Program command to retract
    pcmdAllOff : BOOL;                  // Program command to turn all outputs off
    
    // Operator commands (manual mode only)
    ocmdAdvance : BOOL;                 // Operator command to advance
    ocmdRetract : BOOL;                 // Operator command to retract
    ocmdAllOff : BOOL;                  // Operator command to turn all outputs off
    
    // Reset command (both modes)
    cmdReset : BOOL;                    // Reset fault command
    
    // Permissive inputs (INT with -1 = all OK)
    inPermAdv : INT := -1;              // Advance permissives from field
    inPermRet : INT := -1;              // Retract permissives from field
    
    // Configuration
    cfg : ST_TwoPosActuator_Cfg;        // Configuration structure
END_VAR

VAR_OUTPUT
    EnableOut : BOOL;                   // Enable output
    Status : ST_TwoPosActuator_Sts;     // Status outputs (grouped)
END_VAR

VAR_IN_OUT
    IO : ST_TwoPosActuator_IO;          // IO mapping structure
    HMI : ST_TwoPosActuator_HMI;        // HMI interface
END_VAR

VAR
    // Internal state machine
    currentState : E_TwoPosActuator_State := E_TwoPosActuator_State.Undefined;
    previousState : E_TwoPosActuator_State;
    
    // Timers for motion
    advanceTimer : TON;                 // Advance timeout timer
    retractTimer : TON;                 // Retract timeout timer
    
    // Permissive handlers
    advancePermissives : FB_Permissives;
    retractPermissives : FB_Permissives;
    
    // Command processing
    activeAdvanceCmd : BOOL;            // Active advance command after mode selection
    activeRetractCmd : BOOL;            // Active retract command after mode selection
    activeAllOffCmd : BOOL;             // Active all off command after mode selection
    
    // Edge detection
    rTrigAdvanced : R_TRIG;            // Rising edge for advanced position
    rTrigRetracted : R_TRIG;           // Rising edge for retracted position
    rTrigReset : R_TRIG;               // Rising edge for reset command
    
    // Internal flags
    commandConflict : BOOL;            // TRUE when conflicting commands detected
    bothFeedbackActive : BOOL;         // TRUE when both feedbacks are active
    noFeedbackActive : BOOL;           // TRUE when no feedback is active
    
    // Fault handling
    faultLatched : BOOL;               // Latched fault flag
    lastFault : E_TwoPosActuator_Fault; // Store last fault for diagnostics
END_VAR

//-----------------------------------------------------------------------------
// Main Implementation - FB_TwoPosActuator
//-----------------------------------------------------------------------------
EnableOut := EnableIn;

// Only execute if enabled
IF EnableIn THEN
    
    //-------------------------------------------------------------------------
    // Configuration update from HMI
    //-------------------------------------------------------------------------
    cfg := HMI.cfg;
    
    //-------------------------------------------------------------------------
    // Command Mode Selection and Conflict Detection
    //-------------------------------------------------------------------------
    
    // Select active commands based on working mode
    IF inWorkingMode THEN
        // Automatic mode - only listen to program commands
        activeAdvanceCmd := pcmdAdvance;
        activeRetractCmd := pcmdRetract;
        activeAllOffCmd := pcmdAllOff;
    ELSE
        // Manual mode - listen to operator commands (both input and HMI)
        activeAdvanceCmd := ocmdAdvance OR HMI.ocmdAdvance;
        activeRetractCmd := ocmdRetract OR HMI.ocmdRetract;
        activeAllOffCmd := ocmdAllOff OR HMI.ocmdAllOff;
    END_IF;
    
    // Clear HMI commands after reading (only in manual mode)
    IF NOT inWorkingMode THEN
        IF HMI.ocmdAdvance THEN
            HMI.ocmdAdvance := FALSE;
        END_IF;
        
        IF HMI.ocmdRetract THEN
            HMI.ocmdRetract := FALSE;
        END_IF;
        
        IF HMI.ocmdAllOff THEN
            HMI.ocmdAllOff := FALSE;
        END_IF;
    END_IF;
    
    // Detect conflicting commands (advance and retract cannot be active together)
    commandConflict := activeAdvanceCmd AND activeRetractCmd;
    
    // If conflicting commands detected, clear both and fault
    IF commandConflict THEN
        activeAdvanceCmd := FALSE;
        activeRetractCmd := FALSE;
        activeAllOffCmd := FALSE;
        currentState := E_TwoPosActuator_State.Fault;
        Status.faultCode := E_TwoPosActuator_Fault.ConflictingCommands;
        faultLatched := TRUE;
    END_IF;
    
    // Handle All Off command - overrides other commands and forces safe state
    IF activeAllOffCmd THEN
        activeAdvanceCmd := FALSE;
        activeRetractCmd := FALSE;
        // Note: All Off doesn't change state, just forces outputs off
    END_IF;
    
    //-------------------------------------------------------------------------
    // Permissive Evaluation
    //-------------------------------------------------------------------------
    
    // Advance permissives
    advancePermissives(
        inPermissives := inPermAdv,
        cfg := HMI.advancePerms.cfg
    );
    HMI.advancePerms.sts.OK := advancePermissives.stsOK;
    HMI.advancePerms.sts.PermIntlk := advancePermissives.PermStatus;
    
    // Retract permissives
    retractPermissives(
        inPermissives := inPermRet,
        cfg := HMI.retractPerms.cfg
    );
    HMI.retractPerms.sts.OK := retractPermissives.stsOK;
    HMI.retractPerms.sts.PermIntlk := retractPermissives.PermStatus;
    
    //-------------------------------------------------------------------------
    // Feedback Analysis
    //-------------------------------------------------------------------------
    
    // Analyze feedback conditions
    bothFeedbackActive := IO.inFbkAdvanced AND IO.inFbkRetracted;
    noFeedbackActive := NOT IO.inFbkAdvanced AND NOT IO.inFbkRetracted;
    
    //-------------------------------------------------------------------------
    // Reset Command Processing
    //-------------------------------------------------------------------------
    
    rTrigReset(CLK := cmdReset OR HMI.ocmdReset);
    IF rTrigReset.Q AND faultLatched THEN
        // Clear fault if conditions are safe
        IF NOT commandConflict AND NOT bothFeedbackActive THEN
            faultLatched := FALSE;
            lastFault := Status.faultCode;
            Status.faultCode := E_TwoPosActuator_Fault.None;
            currentState := E_TwoPosActuator_State.Undefined;
        END_IF;
    END_IF;
    
    // Clear HMI reset command
    IF HMI.ocmdReset THEN
        HMI.ocmdReset := FALSE;
    END_IF;
    
    //-------------------------------------------------------------------------
    // State Machine Logic
    //-------------------------------------------------------------------------
    
    // Store previous state for transition detection
    previousState := currentState;
    
    CASE currentState OF
        
        E_TwoPosActuator_State.Undefined:
            //---------------------------------------------------------------------
            // UNDEFINED STATE - Determine initial state based on feedback
            //---------------------------------------------------------------------
            
            // De-energize both outputs in undefined state
            IO.outValveAdvance := FALSE;
            IO.outValveRetract := FALSE;
            
            // Override outputs if All Off command is active
            IF activeAllOffCmd THEN
                IO.outValveAdvance := FALSE;
                IO.outValveRetract := FALSE;
            END_IF;
            
            // Check for fault conditions first
            IF bothFeedbackActive THEN
                currentState := E_TwoPosActuator_State.Fault;
                Status.faultCode := E_TwoPosActuator_Fault.BothFeedbackOn;
                faultLatched := TRUE;
            
            // Determine state based on single feedback
            ELSIF IO.inFbkAdvanced AND NOT IO.inFbkRetracted THEN
                currentState := E_TwoPosActuator_State.Advanced;
            
            ELSIF IO.inFbkRetracted AND NOT IO.inFbkAdvanced THEN
                currentState := E_TwoPosActuator_State.Retracted;
            
            // Handle commands from undefined state with no clear feedback
            ELSIF activeAdvanceCmd AND advancePermissives.stsOK THEN
                currentState := E_TwoPosActuator_State.Advancing;
            
            ELSIF activeRetractCmd AND retractPermissives.stsOK THEN
                currentState := E_TwoPosActuator_State.Retracting;
            
            // Stay in undefined if no feedback and no commands
            END_IF;
        
        E_TwoPosActuator_State.Retracted:
            //---------------------------------------------------------------------
            // RETRACTED STATE
            //---------------------------------------------------------------------
            
            // Handle hold configuration
            IF cfg.cfgHoldAtRetracted AND NOT activeAllOffCmd THEN
                IO.outValveRetract := TRUE;
            ELSE
                IO.outValveRetract := FALSE;
            END_IF;
            IO.outValveAdvance := FALSE;
            
            // Check for fault conditions
            IF bothFeedbackActive THEN
                currentState := E_TwoPosActuator_State.Fault;
                Status.faultCode := E_TwoPosActuator_Fault.BothFeedbackOn;
                faultLatched := TRUE;
            
            ELSIF NOT IO.inFbkRetracted THEN
                currentState := E_TwoPosActuator_State.Fault;
                Status.faultCode := E_TwoPosActuator_Fault.UndefinedState;
                faultLatched := TRUE;
            
            // Handle advance command
            ELSIF activeAdvanceCmd THEN
                IF advancePermissives.stsOK THEN
                    currentState := E_TwoPosActuator_State.Advancing;
                ELSE
                    currentState := E_TwoPosActuator_State.Fault;
                    Status.faultCode := E_TwoPosActuator_Fault.PermissivesNotOK;
                    faultLatched := TRUE;
                END_IF;
            END_IF;
        
        E_TwoPosActuator_State.Advancing:
            //---------------------------------------------------------------------
            // ADVANCING STATE
            //---------------------------------------------------------------------
            
            // Energize advance valve
            IO.outValveAdvance := NOT activeAllOffCmd;
            IO.outValveRetract := FALSE;
            
            // Run advance timer
            advanceTimer(IN := TRUE, PT := DINT_TO_TIME(cfg.cfgAdvTimeoutS * 1000));
            
            // Check for successful advance
            IF IO.inFbkAdvanced AND NOT IO.inFbkRetracted THEN
                currentState := E_TwoPosActuator_State.Advanced;
                advanceTimer(IN := FALSE); // Reset timer
            
            // Check for timeout
            ELSIF advanceTimer.Q THEN
                currentState := E_TwoPosActuator_State.Fault;
                Status.faultCode := E_TwoPosActuator_Fault.AdvanceTimeout;
                faultLatched := TRUE;
                advanceTimer(IN := FALSE); // Reset timer
            
            // Check for fault conditions during motion
            ELSIF bothFeedbackActive THEN
                currentState := E_TwoPosActuator_State.Fault;
                Status.faultCode := E_TwoPosActuator_Fault.BothFeedbackOn;
                faultLatched := TRUE;
                advanceTimer(IN := FALSE); // Reset timer
            
            // Check if permissives are lost during motion
            ELSIF NOT advancePermissives.stsOK THEN
                currentState := E_TwoPosActuator_State.Fault;
                Status.faultCode := E_TwoPosActuator_Fault.PermissivesNotOK;
                faultLatched := TRUE;
                advanceTimer(IN := FALSE); // Reset timer
            END_IF;
        
        E_TwoPosActuator_State.Advanced:
            //---------------------------------------------------------------------
            // ADVANCED STATE
            //---------------------------------------------------------------------
            
            // Handle hold configuration
            IF cfg.cfgHoldAtAdvanced AND NOT activeAllOffCmd THEN
                IO.outValveAdvance := TRUE;
            ELSE
                IO.outValveAdvance := FALSE;
            END_IF;
            IO.outValveRetract := FALSE;
            
            // Check for fault conditions
            IF bothFeedbackActive THEN
                currentState := E_TwoPosActuator_State.Fault;
                Status.faultCode := E_TwoPosActuator_Fault.BothFeedbackOn;
                faultLatched := TRUE;
            
            ELSIF NOT IO.inFbkAdvanced THEN
                currentState := E_TwoPosActuator_State.Fault;
                Status.faultCode := E_TwoPosActuator_Fault.UndefinedState;
                faultLatched := TRUE;
            
            // Handle retract command
            ELSIF activeRetractCmd THEN
                IF retractPermissives.stsOK THEN
                    currentState := E_TwoPosActuator_State.Retracting;
                ELSE
                    currentState := E_TwoPosActuator_State.Fault;
                    Status.faultCode := E_TwoPosActuator_Fault.PermissivesNotOK;
                    faultLatched := TRUE;
                END_IF;
            END_IF;
        
        E_TwoPosActuator_State.Retracting:
            //---------------------------------------------------------------------
            // RETRACTING STATE
            //---------------------------------------------------------------------
            
            // Energize retract valve
            IO.outValveRetract := NOT activeAllOffCmd;
            IO.outValveAdvance := FALSE;
            
            // Run retract timer
            retractTimer(IN := TRUE, PT := DINT_TO_TIME(cfg.cfgRetTimeoutS * 1000));
            
            // Check for successful retract
            IF IO.inFbkRetracted AND NOT IO.inFbkAdvanced THEN
                currentState := E_TwoPosActuator_State.Retracted;
                retractTimer(IN := FALSE); // Reset timer
            
            // Check for timeout
            ELSIF retractTimer.Q THEN
                currentState := E_TwoPosActuator_State.Fault;
                Status.faultCode := E_TwoPosActuator_Fault.RetractTimeout;
                faultLatched := TRUE;
                retractTimer(IN := FALSE); // Reset timer
            
            // Check for fault conditions during motion
            ELSIF bothFeedbackActive THEN
                currentState := E_TwoPosActuator_State.Fault;
                Status.faultCode := E_TwoPosActuator_Fault.BothFeedbackOn;
                faultLatched := TRUE;
                retractTimer(IN := FALSE); // Reset timer
            
            // Check if permissives are lost during motion
            ELSIF NOT retractPermissives.stsOK THEN
                currentState := E_TwoPosActuator_State.Fault;
                Status.faultCode := E_TwoPosActuator_Fault.PermissivesNotOK;
                faultLatched := TRUE;
                retractTimer(IN := FALSE); // Reset timer
            END_IF;
        
        E_TwoPosActuator_State.Fault:
            //---------------------------------------------------------------------
            // FAULT STATE
            //---------------------------------------------------------------------
            
            // De-energize both outputs in fault state
            IO.outValveAdvance := FALSE;
            IO.outValveRetract := FALSE;
            
            // Stop timers
            advanceTimer(IN := FALSE);
            retractTimer(IN := FALSE);
            
            // Fault is cleared by reset command (handled above)
    END_CASE;
    
    //-------------------------------------------------------------------------
    // Status Output Generation
    //-------------------------------------------------------------------------
    
    // Update status structure
    Status.state := currentState;
    Status.stsAdvanced := (currentState = E_TwoPosActuator_State.Advanced);
    Status.stsRetracted := (currentState = E_TwoPosActuator_State.Retracted);
    Status.stsMoving := (currentState = E_TwoPosActuator_State.Advancing) OR 
                       (currentState = E_TwoPosActuator_State.Retracting);
    Status.stsFaulted := (currentState = E_TwoPosActuator_State.Fault) OR faultLatched;
    Status.lastFaultCode := lastFault;
    
    // Generate one-shots for position reached
    rTrigAdvanced(CLK := Status.stsAdvanced);
    Status.osAdvanced := rTrigAdvanced.Q;
    
    rTrigRetracted(CLK := Status.stsRetracted);
    Status.osRetracted := rTrigRetracted.Q;
    
    //-------------------------------------------------------------------------
    // HMI Status Update
    //-------------------------------------------------------------------------
    
    // Copy status to HMI
    HMI.sts := Status;
    
    // Generate human-readable state string
    CASE currentState OF
        E_TwoPosActuator_State.Undefined:
            HMI.stateString := 'Undefined';
        E_TwoPosActuator_State.Retracted:
            HMI.stateString := 'Retracted';
        E_TwoPosActuator_State.Advancing:
            HMI.stateString := 'Advancing';
        E_TwoPosActuator_State.Advanced:
            HMI.stateString := 'Advanced';
        E_TwoPosActuator_State.Retracting:
            HMI.stateString := 'Retracting';
        E_TwoPosActuator_State.Fault:
            HMI.stateString := 'Fault';
    ELSE
        HMI.stateString := 'Unknown';
    END_CASE;
    
    // Generate human-readable fault string
    CASE Status.faultCode OF
        E_TwoPosActuator_Fault.None:
            HMI.faultString := 'No Fault';
        E_TwoPosActuator_Fault.AdvanceTimeout:
            HMI.faultString := 'Advance Timeout';
        E_TwoPosActuator_Fault.RetractTimeout:
            HMI.faultString := 'Retract Timeout';
        E_TwoPosActuator_Fault.BothFeedbackOn:
            HMI.faultString := 'Both Feedbacks Active';
        E_TwoPosActuator_Fault.UndefinedState:
            HMI.faultString := 'Position Undefined';
        E_TwoPosActuator_Fault.PermissivesNotOK:
            HMI.faultString := 'Permissives Not OK';
        E_TwoPosActuator_Fault.ConflictingCommands:
            HMI.faultString := 'Conflicting Commands';
        E_TwoPosActuator_Fault.NoFeedback:
            HMI.faultString := 'No Position Feedback';
    ELSE
        HMI.faultString := 'Unknown Fault';
    END_CASE;
    
    // Generate human-readable last fault string
    CASE Status.lastFaultCode OF
        E_TwoPosActuator_Fault.None:
            HMI.lastFaultString := 'No Previous Fault';
        E_TwoPosActuator_Fault.AdvanceTimeout:
            HMI.lastFaultString := 'Last: Advance Timeout';
        E_TwoPosActuator_Fault.RetractTimeout:
            HMI.lastFaultString := 'Last: Retract Timeout';
        E_TwoPosActuator_Fault.BothFeedbackOn:
            HMI.lastFaultString := 'Last: Both Feedbacks Active';
        E_TwoPosActuator_Fault.UndefinedState:
            HMI.lastFaultString := 'Last: Position Undefined';
        E_TwoPosActuator_Fault.PermissivesNotOK:
            HMI.lastFaultString := 'Last: Permissives Not OK';
        E_TwoPosActuator_Fault.ConflictingCommands:
            HMI.lastFaultString := 'Last: Conflicting Commands';
        E_TwoPosActuator_Fault.NoFeedback:
            HMI.lastFaultString := 'Last: No Position Feedback';
    ELSE
        HMI.lastFaultString := 'Last: Unknown Fault';
    END_CASE;
    
ELSE
    // Disabled - de-energize outputs and reset timers
    IO.outValveAdvance := FALSE;
    IO.outValveRetract := FALSE;
    advanceTimer(IN := FALSE);
    retractTimer(IN := FALSE);
END_IF;

END_FUNCTION_BLOCK
